// TIA Portal V16 export
// export: Created 2023-03-29T11:04:27.7848661Z, ExportSetting WithDefaults, DisplayName Totally Integrated Automation Portal, DisplayVersion V16 Update 6, DisplayName TIA Portal Version Control Interface, DisplayVersion V16 Update 2, DisplayName TIA Portal Openness, DisplayVersion V16 Update 6, DisplayName STEP 7 Professional, DisplayVersion V16 Update 6, DisplayName STEP 7 Safety, DisplayVersion V16, DisplayName WinCC Advanced, DisplayVersion V16 Update 6
ORGANIZATION_BLOCK "Startup"   // OB100, LAD, Startup
TITLE = "Complete Restart"
{ S7_Optimized_Access := 'TRUE' }
AUTHOR : RTecmer
VERSION : 0.1
// stored: AutoNumber true, IsIECCheckEnabled false, SetENOAutomatically false
   VAR_INPUT
      LostRetentive : Bool;   // True if retentive data are lost
      LostRTC : Bool;   // True if date and time are lost
   END_VAR
BEGIN

REGION Network 1: inicjacja master modbus RTU / Incjalizacja modułu Master CM1241 (RS485) Modbus RTU
   // Komunikacja z przepływomierzami MP04 i falownikiem Danfoss
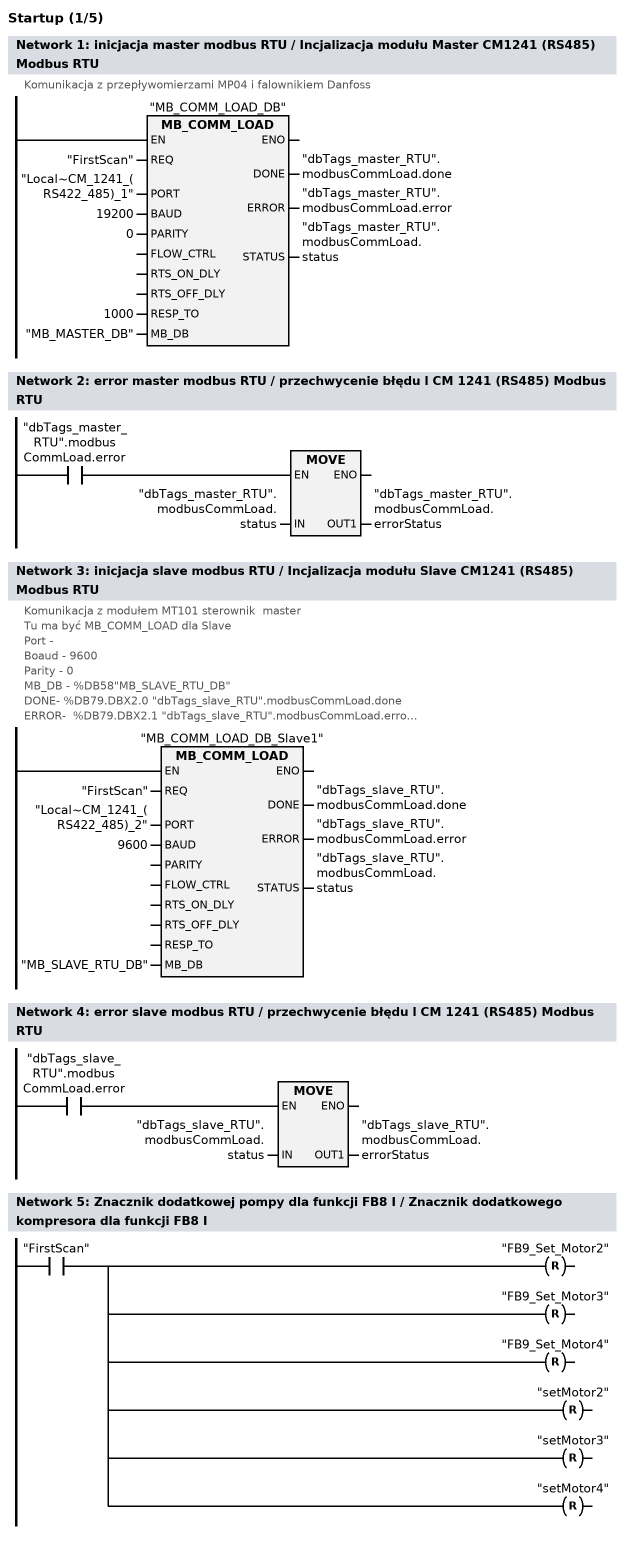
   RUNG wire#powerrail
      "MB_COMM_LOAD_DB".MB_COMM_LOAD(REQ := "FirstScan", PORT := "Local~CM_1241_(RS422_485)_1", BAUD := 19200, PARITY := 0, FLOW_CTRL :=, RTS_ON_DLY :=, RTS_OFF_DLY :=, RESP_TO := 1000, MB_DB := "MB_MASTER_DB", DONE => "dbTags_master_RTU".modbusCommLoad.done, ERROR => "dbTags_master_RTU".modbusCommLoad.error, STATUS => "dbTags_master_RTU".modbusCommLoad.status)
   END_RUNG
   // the same network as SCL:
   "MB_COMM_LOAD_DB"(REQ := "FirstScan",   // MB_COMM_LOAD
                     PORT := "Local~CM_1241_(RS422_485)_1",
                     BAUD := 19200,
                     PARITY := 0,
                     RESP_TO := 1000,
                     MB_DB := "MB_MASTER_DB",
                     DONE => "dbTags_master_RTU".modbusCommLoad.done,
                     ERROR => "dbTags_master_RTU".modbusCommLoad.error,
                     STATUS => "dbTags_master_RTU".modbusCommLoad.status);
END_REGION

REGION Network 2: error master modbus RTU / przechwycenie błędu l CM 1241 (RS485) Modbus RTU
   RUNG wire#powerrail
      Contact( "dbTags_master_RTU".modbusCommLoad.error )
      { S7_GenerateENO := "TRUE" } Move(in := "dbTags_master_RTU".modbusCommLoad.status, out1 => "dbTags_master_RTU".modbusCommLoad.errorStatus)
   END_RUNG
   // the same network as SCL:
   IF "dbTags_master_RTU".modbusCommLoad.error THEN
       "dbTags_master_RTU".modbusCommLoad.errorStatus := "dbTags_master_RTU".modbusCommLoad.status;
   END_IF;
END_REGION

REGION Network 3: inicjacja slave modbus RTU / Incjalizacja modułu Slave CM1241 (RS485) Modbus RTU
   // Komunikacja z modułem MT101 sterownik  master
   // 
   // Tu ma być MB_COMM_LOAD dla Slave
   // Port -
   // Boaud - 9600
   // Parity - 0
   // MB_DB - %DB58"MB_SLAVE_RTU_DB"
   // DONE- %DB79.DBX2.0 "dbTags_slave_RTU".modbusCommLoad.done
   // ERROR-  %DB79.DBX2.1 "dbTags_slave_RTU".modbusCommLoad.error
   // STATUS - %DB79.DBX2.2 "dbTags_slave_RTU".modbusCommLoad.status
   RUNG wire#powerrail
      "MB_COMM_LOAD_DB_Slave1".MB_COMM_LOAD(REQ := "FirstScan", PORT := "Local~CM_1241_(RS422_485)_2", BAUD := 9600, PARITY :=, FLOW_CTRL :=, RTS_ON_DLY :=, RTS_OFF_DLY :=, RESP_TO :=, MB_DB := "MB_SLAVE_RTU_DB", DONE => "dbTags_slave_RTU".modbusCommLoad.done, ERROR => "dbTags_slave_RTU".modbusCommLoad.error, STATUS => "dbTags_slave_RTU".modbusCommLoad.status)
   END_RUNG
   // the same network as SCL:
   "MB_COMM_LOAD_DB_Slave1"(REQ := "FirstScan",   // MB_COMM_LOAD
                           PORT := "Local~CM_1241_(RS422_485)_2",
                           BAUD := 9600,
                           MB_DB := "MB_SLAVE_RTU_DB",
                           DONE => "dbTags_slave_RTU".modbusCommLoad.done,
                           ERROR => "dbTags_slave_RTU".modbusCommLoad.error,
                           STATUS => "dbTags_slave_RTU".modbusCommLoad.status);
END_REGION

REGION Network 4: error slave modbus RTU / przechwycenie błędu l CM 1241 (RS485) Modbus RTU
   RUNG wire#powerrail
      Contact( "dbTags_slave_RTU".modbusCommLoad.error )
      { S7_GenerateENO := "TRUE" } Move(in := "dbTags_slave_RTU".modbusCommLoad.status, out1 => "dbTags_slave_RTU".modbusCommLoad.errorStatus)
   END_RUNG
   // the same network as SCL:
   IF "dbTags_slave_RTU".modbusCommLoad.error THEN
       "dbTags_slave_RTU".modbusCommLoad.errorStatus := "dbTags_slave_RTU".modbusCommLoad.status;
   END_IF;
END_REGION

REGION Network 5: Znacznik dodatkowej pompy dla funkcji FB8 I / Znacznik dodatkowego kompresora dla funkcji FB8 I
   RUNG wire#powerrail
      Contact( "FirstScan" )
      wire#w1
      R_Coil( "FB9_Set_Motor2" )
   END_RUNG
   RUNG wire#w1
      R_Coil( "FB9_Set_Motor3" )
   END_RUNG
   RUNG wire#w1
      R_Coil( "FB9_Set_Motor4" )
   END_RUNG
   RUNG wire#w1
      R_Coil( "setMotor2" )
   END_RUNG
   RUNG wire#w1
      R_Coil( "setMotor3" )
   END_RUNG
   RUNG wire#w1
      R_Coil( "setMotor4" )
   END_RUNG
   // the same network as SCL:
   IF "FirstScan" THEN
       "FB9_Set_Motor2" := FALSE;
       "FB9_Set_Motor3" := FALSE;
       "FB9_Set_Motor4" := FALSE;
       "setMotor2" := FALSE;
       "setMotor3" := FALSE;
       "setMotor4" := FALSE;
   END_IF;
END_REGION

REGION Network 6
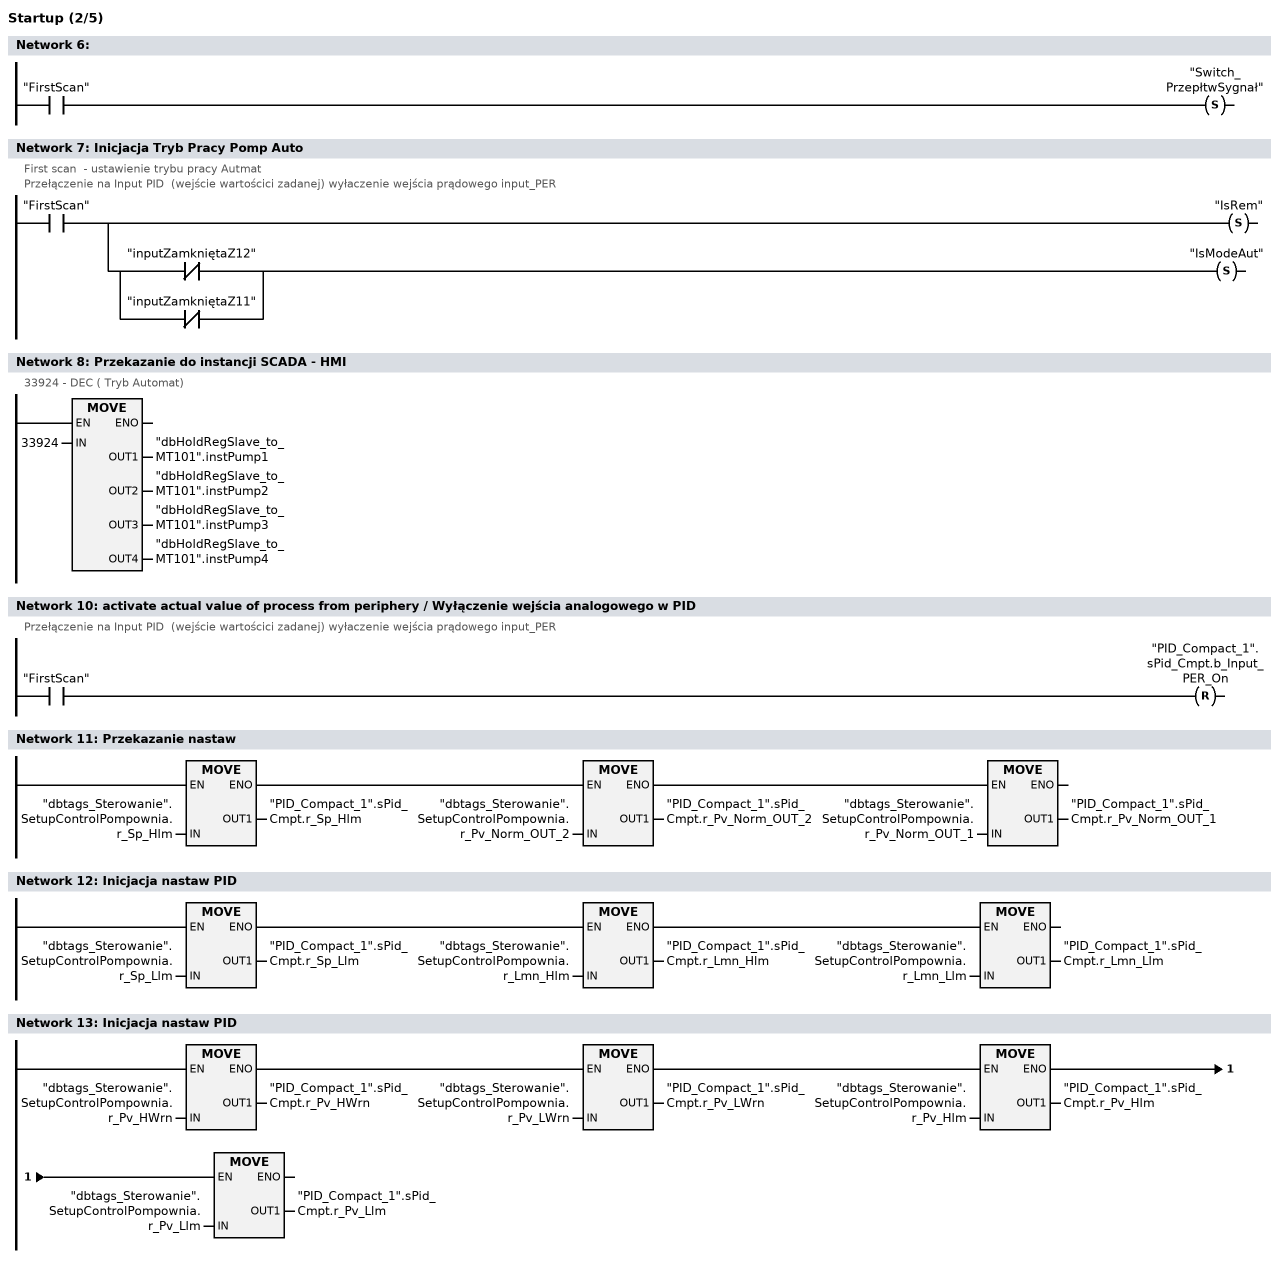
   RUNG wire#powerrail
      Contact( "FirstScan" )
      S_Coil( "Switch_PrzepłtwSygnał" )
   END_RUNG
   // the same network as SCL:
   IF "FirstScan" THEN "Switch_PrzepłtwSygnał" := TRUE; END_IF;
END_REGION

REGION Network 7: Inicjacja Tryb Pracy Pomp Auto
   // First scan  - ustawienie trybu pracy Autmat 
   // Przełączenie na Input PID  (wejście wartościci zadanej) wyłaczenie wejścia prądowego input_PER
   RUNG wire#powerrail
      Contact( "FirstScan" )
      wire#w1
      S_Coil( "IsRem" )
   END_RUNG
   RUNG wire#w1
      I_Contact( "inputZamkniętaZ12" )
      wire#w2
      S_Coil( "IsModeAut" )
   END_RUNG
   RUNG wire#w1
      I_Contact( "inputZamkniętaZ11" )
   END_RUNG wire#w2
   // the same network as SCL:
   IF "FirstScan" THEN "IsRem" := TRUE; END_IF;
   IF "FirstScan" AND (NOT "inputZamkniętaZ12" OR NOT "inputZamkniętaZ11") THEN "IsModeAut" := TRUE; END_IF;
END_REGION

REGION Network 8: Przekazanie do instancji SCADA - HMI
   // 33924 - DEC ( Tryb Automat)
   RUNG wire#powerrail
      { S7_GenerateENO := "TRUE" } Move(in := 33924, out1 => "dbHoldRegSlave_to_MT101".instPump1, out2 => "dbHoldRegSlave_to_MT101".instPump2, out3 => "dbHoldRegSlave_to_MT101".instPump3, out4 => "dbHoldRegSlave_to_MT101".instPump4)
   END_RUNG
   // the same network as SCL:
   "dbHoldRegSlave_to_MT101".instPump1 := 33924;
   "dbHoldRegSlave_to_MT101".instPump2 := 33924;
   "dbHoldRegSlave_to_MT101".instPump3 := 33924;
   "dbHoldRegSlave_to_MT101".instPump4 := 33924;
END_REGION

REGION Network 10: activate actual value of process from periphery / Wyłączenie wejścia analogowego w PID
   // Przełączenie na Input PID  (wejście wartościci zadanej) wyłaczenie wejścia prądowego input_PER
   RUNG wire#powerrail
      Contact( "FirstScan" )
      R_Coil( "PID_Compact_1".sPid_Cmpt.b_Input_PER_On )
   END_RUNG
   // the same network as SCL:
   IF "FirstScan" THEN "PID_Compact_1".sPid_Cmpt.b_Input_PER_On := FALSE; END_IF;
END_REGION

REGION Network 11: Przekazanie nastaw
   RUNG wire#powerrail
      { S7_GenerateENO := "TRUE" } Move(in := "dbtags_Sterowanie".SetupControlPompownia.r_Sp_Hlm, out1 => "PID_Compact_1".sPid_Cmpt.r_Sp_Hlm)
      { S7_GenerateENO := "TRUE" } Move(in := "dbtags_Sterowanie".SetupControlPompownia.r_Pv_Norm_OUT_2, out1 => "PID_Compact_1".sPid_Cmpt.r_Pv_Norm_OUT_2)
      { S7_GenerateENO := "TRUE" } Move(in := "dbtags_Sterowanie".SetupControlPompownia.r_Pv_Norm_OUT_1, out1 => "PID_Compact_1".sPid_Cmpt.r_Pv_Norm_OUT_1)
   END_RUNG
   // the same network as SCL:
   // ENO of a box is taken as its EN; it also drops when the box reports an error
   "PID_Compact_1".sPid_Cmpt.r_Sp_Hlm := "dbtags_Sterowanie".SetupControlPompownia.r_Sp_Hlm;
   "PID_Compact_1".sPid_Cmpt.r_Pv_Norm_OUT_2 := "dbtags_Sterowanie".SetupControlPompownia.r_Pv_Norm_OUT_2;
   "PID_Compact_1".sPid_Cmpt.r_Pv_Norm_OUT_1 := "dbtags_Sterowanie".SetupControlPompownia.r_Pv_Norm_OUT_1;
END_REGION

REGION Network 12: Inicjacja nastaw PID
   RUNG wire#powerrail
      { S7_GenerateENO := "TRUE" } Move(in := "dbtags_Sterowanie".SetupControlPompownia.r_Sp_Llm, out1 => "PID_Compact_1".sPid_Cmpt.r_Sp_Llm)
      { S7_GenerateENO := "TRUE" } Move(in := "dbtags_Sterowanie".SetupControlPompownia.r_Lmn_Hlm, out1 => "PID_Compact_1".sPid_Cmpt.r_Lmn_Hlm)
      { S7_GenerateENO := "TRUE" } Move(in := "dbtags_Sterowanie".SetupControlPompownia.r_Lmn_Llm, out1 => "PID_Compact_1".sPid_Cmpt.r_Lmn_Llm)
   END_RUNG
   // the same network as SCL:
   // ENO of a box is taken as its EN; it also drops when the box reports an error
   "PID_Compact_1".sPid_Cmpt.r_Sp_Llm := "dbtags_Sterowanie".SetupControlPompownia.r_Sp_Llm;
   "PID_Compact_1".sPid_Cmpt.r_Lmn_Hlm := "dbtags_Sterowanie".SetupControlPompownia.r_Lmn_Hlm;
   "PID_Compact_1".sPid_Cmpt.r_Lmn_Llm := "dbtags_Sterowanie".SetupControlPompownia.r_Lmn_Llm;
END_REGION

REGION Network 13: Inicjacja nastaw PID
   RUNG wire#powerrail
      { S7_GenerateENO := "TRUE" } Move(in := "dbtags_Sterowanie".SetupControlPompownia.r_Pv_HWrn, out1 => "PID_Compact_1".sPid_Cmpt.r_Pv_HWrn)
      { S7_GenerateENO := "TRUE" } Move(in := "dbtags_Sterowanie".SetupControlPompownia.r_Pv_LWrn, out1 => "PID_Compact_1".sPid_Cmpt.r_Pv_LWrn)
      { S7_GenerateENO := "TRUE" } Move(in := "dbtags_Sterowanie".SetupControlPompownia.r_Pv_Hlm, out1 => "PID_Compact_1".sPid_Cmpt.r_Pv_Hlm)
      { S7_GenerateENO := "TRUE" } Move(in := "dbtags_Sterowanie".SetupControlPompownia.r_Pv_Llm, out1 => "PID_Compact_1".sPid_Cmpt.r_Pv_Llm)
   END_RUNG
   // the same network as SCL:
   // ENO of a box is taken as its EN; it also drops when the box reports an error
   "PID_Compact_1".sPid_Cmpt.r_Pv_HWrn := "dbtags_Sterowanie".SetupControlPompownia.r_Pv_HWrn;
   "PID_Compact_1".sPid_Cmpt.r_Pv_LWrn := "dbtags_Sterowanie".SetupControlPompownia.r_Pv_LWrn;
   "PID_Compact_1".sPid_Cmpt.r_Pv_Hlm := "dbtags_Sterowanie".SetupControlPompownia.r_Pv_Hlm;
   "PID_Compact_1".sPid_Cmpt.r_Pv_Llm := "dbtags_Sterowanie".SetupControlPompownia.r_Pv_Llm;
END_REGION

REGION Network 14: Zasuwa Z11 Tryb Automat
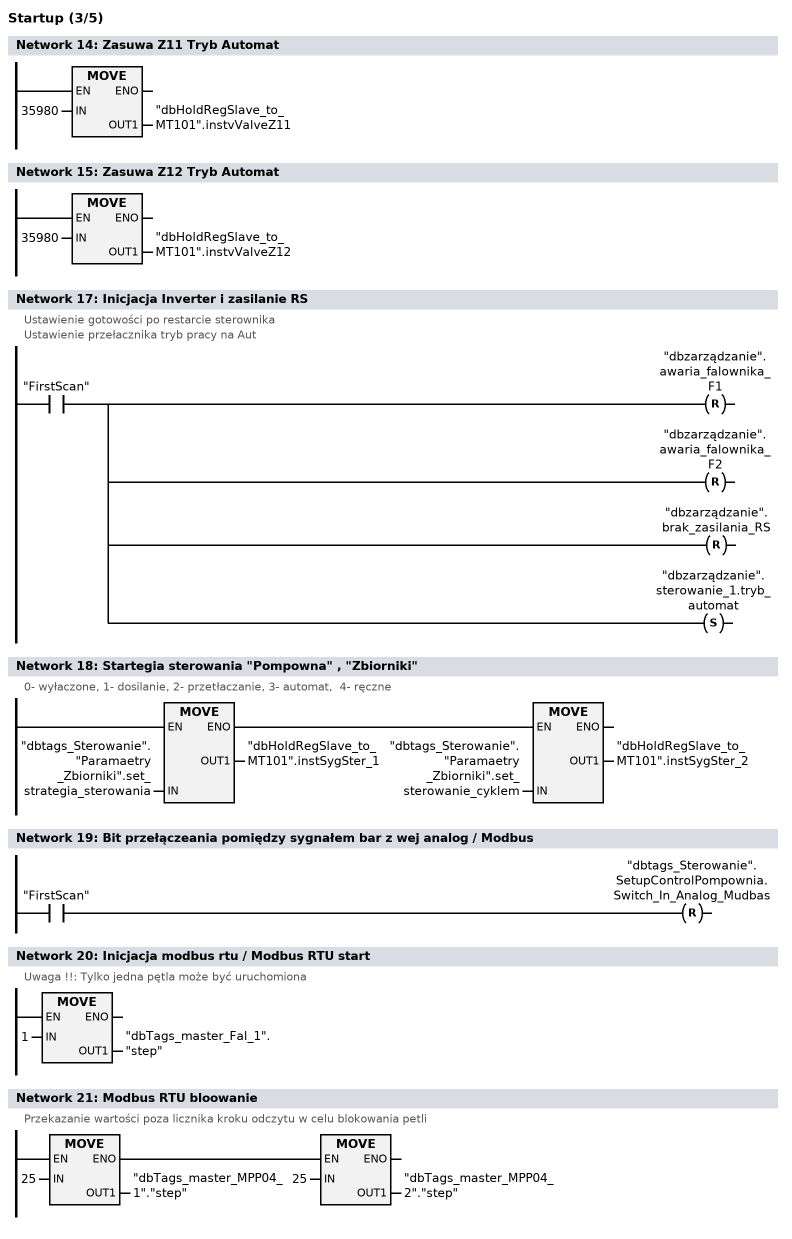
   RUNG wire#powerrail
      Move(in := 35980, out1 => "dbHoldRegSlave_to_MT101".instvValveZ11)
   END_RUNG
   // the same network as SCL:
   "dbHoldRegSlave_to_MT101".instvValveZ11 := 35980;
END_REGION

REGION Network 15: Zasuwa Z12 Tryb Automat
   RUNG wire#powerrail
      Move(in := 35980, out1 => "dbHoldRegSlave_to_MT101".instvValveZ12)
   END_RUNG
   // the same network as SCL:
   "dbHoldRegSlave_to_MT101".instvValveZ12 := 35980;
END_REGION

REGION Network 17: Inicjacja Inverter i zasilanie RS
   // Ustawienie gotowości po restarcie sterownika
   // Ustawienie przełacznika tryb pracy na Aut
   RUNG wire#powerrail
      Contact( "FirstScan" )
      wire#w1
      R_Coil( "dbzarządzanie".awaria_falownika_F1 )
   END_RUNG
   RUNG wire#w1
      R_Coil( "dbzarządzanie".awaria_falownika_F2 )
   END_RUNG
   RUNG wire#w1
      R_Coil( "dbzarządzanie".brak_zasilania_RS )
   END_RUNG
   RUNG wire#w1
      S_Coil( "dbzarządzanie".sterowanie_1.tryb_automat )
   END_RUNG
   // the same network as SCL:
   IF "FirstScan" THEN
       "dbzarządzanie".awaria_falownika_F1 := FALSE;
       "dbzarządzanie".awaria_falownika_F2 := FALSE;
       "dbzarządzanie".brak_zasilania_RS := FALSE;
       "dbzarządzanie".sterowanie_1.tryb_automat := TRUE;
   END_IF;
END_REGION

REGION Network 18: Startegia sterowania "Pompowna" , "Zbiorniki"
   // 0- wyłaczone, 1- dosilanie, 2- przetłaczanie, 3- automat,  4- ręczne
   RUNG wire#powerrail
      Move(in := "dbtags_Sterowanie"."Paramaetry _Zbiorniki".set_strategia_sterowania, out1 => "dbHoldRegSlave_to_MT101".instSygSter_1)
      Move(in := "dbtags_Sterowanie"."Paramaetry _Zbiorniki".set_sterowanie_cyklem, out1 => "dbHoldRegSlave_to_MT101".instSygSter_2)
   END_RUNG
   // the same network as SCL:
   "dbHoldRegSlave_to_MT101".instSygSter_1 := "dbtags_Sterowanie"."Paramaetry _Zbiorniki".set_strategia_sterowania;
   "dbHoldRegSlave_to_MT101".instSygSter_2 := "dbtags_Sterowanie"."Paramaetry _Zbiorniki".set_sterowanie_cyklem;
END_REGION

REGION Network 19: Bit przełączeania pomiędzy sygnałem bar z wej analog / Modbus
   RUNG wire#powerrail
      Contact( "FirstScan" )
      R_Coil( "dbtags_Sterowanie".SetupControlPompownia.Switch_In_Analog_Mudbas )
   END_RUNG
   // the same network as SCL:
   IF "FirstScan" THEN "dbtags_Sterowanie".SetupControlPompownia.Switch_In_Analog_Mudbas := FALSE; END_IF;
END_REGION

REGION Network 20: Inicjacja modbus rtu / Modbus RTU start
   // Uwaga !!: Tylko jedna pętla może być uruchomiona
   RUNG wire#powerrail
      { S7_GenerateENO := "TRUE" } Move(in := 1, out1 => "dbTags_master_Fal_1"."step")
   END_RUNG
   // the same network as SCL:
   "dbTags_master_Fal_1"."step" := 1;
END_REGION

REGION Network 21: Modbus RTU bloowanie
   // Przekazanie wartości poza licznika kroku odczytu w celu blokowania petli
   RUNG wire#powerrail
      { S7_GenerateENO := "TRUE" } Move(in := 25, out1 => "dbTags_master_MPP04_1"."step")
      { S7_GenerateENO := "TRUE" } Move(in := 25, out1 => "dbTags_master_MPP04_2"."step")
   END_RUNG
   // the same network as SCL:
   // ENO of a box is taken as its EN; it also drops when the box reports an error
   "dbTags_master_MPP04_1"."step" := 25;
   "dbTags_master_MPP04_2"."step" := 25;
END_REGION

REGION Network 22: Przełącznik wyboru źródła zadawania wartości granicznej dopuszczalnego prądy falownika
   // 1 - zadawany w konfiguracju z HMI
   // 0 - odczytany z falownika
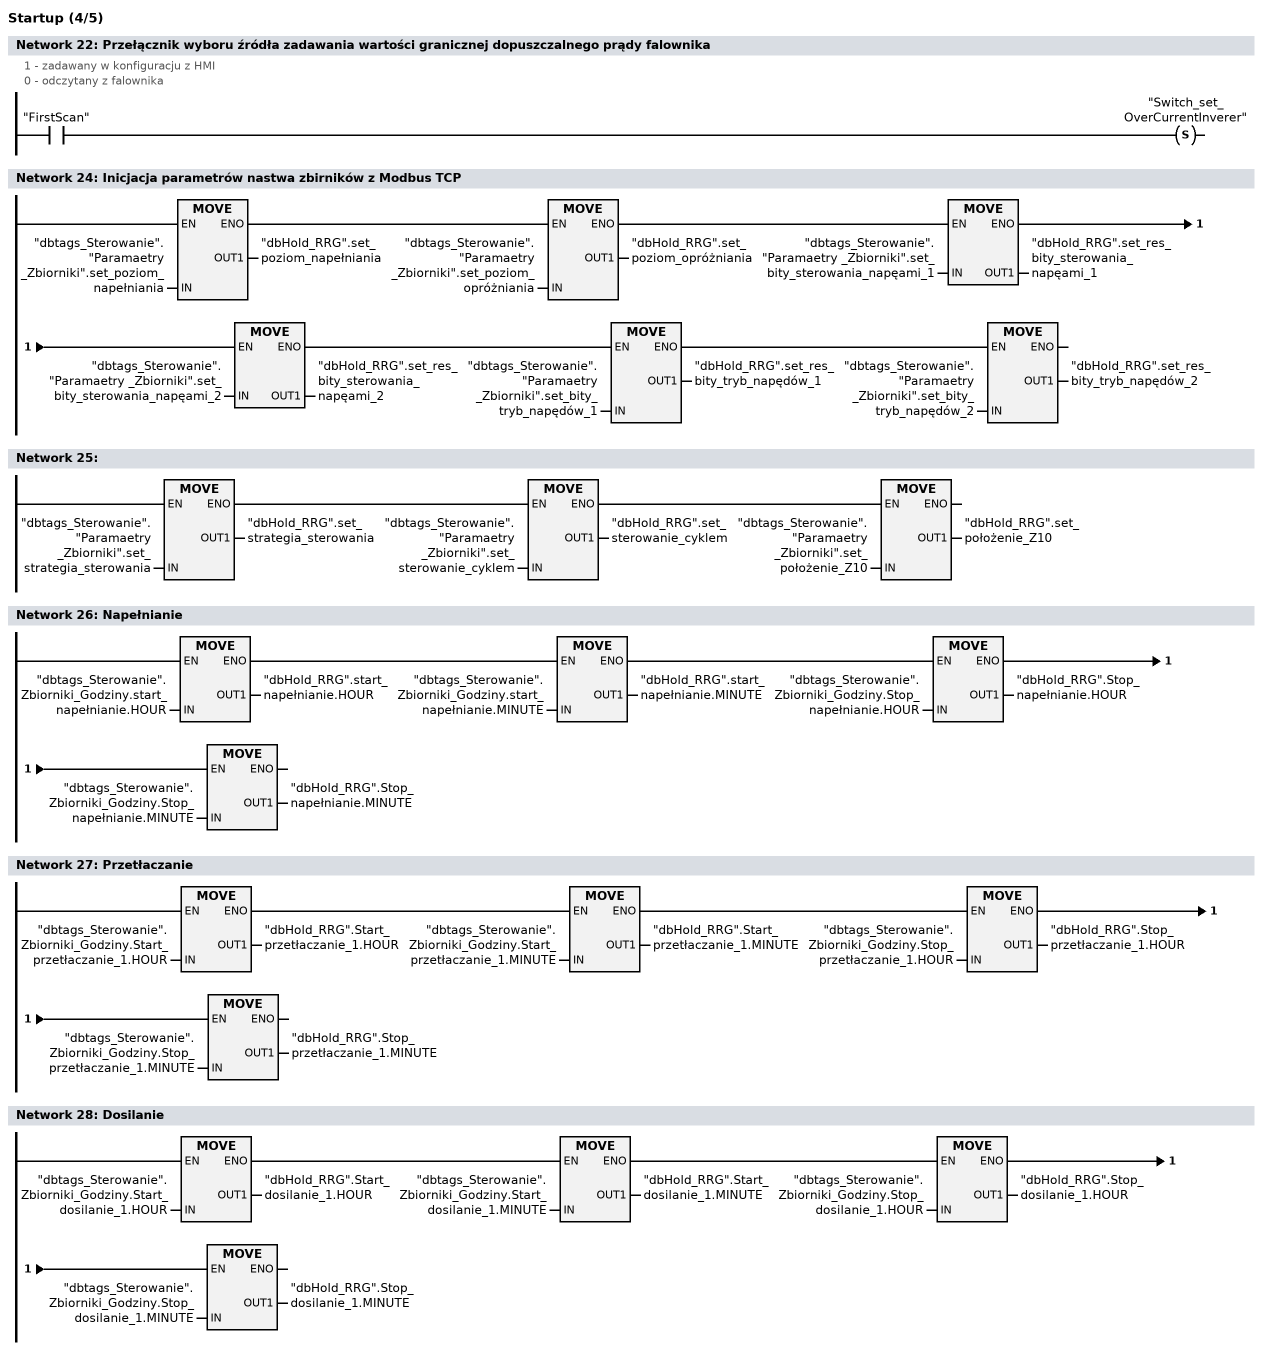
   RUNG wire#powerrail
      Contact( "FirstScan" )
      S_Coil( "Switch_set_OverCurrentInverer" )
   END_RUNG
   // the same network as SCL:
   IF "FirstScan" THEN "Switch_set_OverCurrentInverer" := TRUE; END_IF;
END_REGION

REGION Network 23 (SCL): Ustawienie Setpoint SV do regulatora
   // Wartość ciśnienia zadanego zależna od wybranej strategii
   CASE "dbHoldRegSlave_to_MT101".instSygSter_1 OF
     1:
       "dbdane".Setpoint_SV := "dbtags_Sterowanie".SetupControlPompownia.set_barDN500_B5 ;
     2:
       "dbdane".Setpoint_SV := "dbtags_Sterowanie".SetupControlPompownia.set_barDN225_B6;
     3:
       "dbdane".Setpoint_SV := "dbdane".Setpoint_bar_automat ;

     ELSE
       "dbdane".Setpoint_SV := 0.0;
       ;
   END_CASE;
END_REGION

REGION Network 24: Inicjacja parametrów nastwa zbirników z Modbus TCP
   RUNG wire#powerrail
      Move(in := "dbtags_Sterowanie"."Paramaetry _Zbiorniki".set_poziom_napełniania, out1 => "dbHold_RRG".set_poziom_napełniania)
      Move(in := "dbtags_Sterowanie"."Paramaetry _Zbiorniki".set_poziom_opróżniania, out1 => "dbHold_RRG".set_poziom_opróżniania)
      Move(in := "dbtags_Sterowanie"."Paramaetry _Zbiorniki".set_bity_sterowania_napęami_1, out1 => "dbHold_RRG".set_res_bity_sterowania_napęami_1)
      Move(in := "dbtags_Sterowanie"."Paramaetry _Zbiorniki".set_bity_sterowania_napęami_2, out1 => "dbHold_RRG".set_res_bity_sterowania_napęami_2)
      Move(in := "dbtags_Sterowanie"."Paramaetry _Zbiorniki".set_bity_tryb_napędów_1, out1 => "dbHold_RRG".set_res_bity_tryb_napędów_1)
      Move(in := "dbtags_Sterowanie"."Paramaetry _Zbiorniki".set_bity_tryb_napędów_2, out1 => "dbHold_RRG".set_res_bity_tryb_napędów_2)
   END_RUNG
   // the same network as SCL:
   "dbHold_RRG".set_poziom_napełniania := "dbtags_Sterowanie"."Paramaetry _Zbiorniki".set_poziom_napełniania;
   "dbHold_RRG".set_poziom_opróżniania := "dbtags_Sterowanie"."Paramaetry _Zbiorniki".set_poziom_opróżniania;
   "dbHold_RRG".set_res_bity_sterowania_napęami_1 := "dbtags_Sterowanie"."Paramaetry _Zbiorniki".set_bity_sterowania_napęami_1;
   "dbHold_RRG".set_res_bity_sterowania_napęami_2 := "dbtags_Sterowanie"."Paramaetry _Zbiorniki".set_bity_sterowania_napęami_2;
   "dbHold_RRG".set_res_bity_tryb_napędów_1 := "dbtags_Sterowanie"."Paramaetry _Zbiorniki".set_bity_tryb_napędów_1;
   "dbHold_RRG".set_res_bity_tryb_napędów_2 := "dbtags_Sterowanie"."Paramaetry _Zbiorniki".set_bity_tryb_napędów_2;
END_REGION

REGION Network 25
   RUNG wire#powerrail
      Move(in := "dbtags_Sterowanie"."Paramaetry _Zbiorniki".set_strategia_sterowania, out1 => "dbHold_RRG".set_strategia_sterowania)
      Move(in := "dbtags_Sterowanie"."Paramaetry _Zbiorniki".set_sterowanie_cyklem, out1 => "dbHold_RRG".set_sterowanie_cyklem)
      Move(in := "dbtags_Sterowanie"."Paramaetry _Zbiorniki".set_położenie_Z10, out1 => "dbHold_RRG".set_położenie_Z10)
   END_RUNG
   // the same network as SCL:
   "dbHold_RRG".set_strategia_sterowania := "dbtags_Sterowanie"."Paramaetry _Zbiorniki".set_strategia_sterowania;
   "dbHold_RRG".set_sterowanie_cyklem := "dbtags_Sterowanie"."Paramaetry _Zbiorniki".set_sterowanie_cyklem;
   "dbHold_RRG".set_położenie_Z10 := "dbtags_Sterowanie"."Paramaetry _Zbiorniki".set_położenie_Z10;
END_REGION

REGION Network 26: Napełnianie
   RUNG wire#powerrail
      Move(in := "dbtags_Sterowanie".Zbiorniki_Godziny.start_napełnianie.HOUR, out1 => "dbHold_RRG".start_napełnianie.HOUR)
      Move(in := "dbtags_Sterowanie".Zbiorniki_Godziny.start_napełnianie.MINUTE, out1 => "dbHold_RRG".start_napełnianie.MINUTE)
      Move(in := "dbtags_Sterowanie".Zbiorniki_Godziny.Stop_napełnianie.HOUR, out1 => "dbHold_RRG".Stop_napełnianie.HOUR)
      Move(in := "dbtags_Sterowanie".Zbiorniki_Godziny.Stop_napełnianie.MINUTE, out1 => "dbHold_RRG".Stop_napełnianie.MINUTE)
   END_RUNG
   // the same network as SCL:
   "dbHold_RRG".start_napełnianie.HOUR := "dbtags_Sterowanie".Zbiorniki_Godziny.start_napełnianie.HOUR;
   "dbHold_RRG".start_napełnianie.MINUTE := "dbtags_Sterowanie".Zbiorniki_Godziny.start_napełnianie.MINUTE;
   "dbHold_RRG".Stop_napełnianie.HOUR := "dbtags_Sterowanie".Zbiorniki_Godziny.Stop_napełnianie.HOUR;
   "dbHold_RRG".Stop_napełnianie.MINUTE := "dbtags_Sterowanie".Zbiorniki_Godziny.Stop_napełnianie.MINUTE;
END_REGION

REGION Network 27: Przetłaczanie
   RUNG wire#powerrail
      Move(in := "dbtags_Sterowanie".Zbiorniki_Godziny.Start_przetłaczanie_1.HOUR, out1 => "dbHold_RRG".Start_przetłaczanie_1.HOUR)
      Move(in := "dbtags_Sterowanie".Zbiorniki_Godziny.Start_przetłaczanie_1.MINUTE, out1 => "dbHold_RRG".Start_przetłaczanie_1.MINUTE)
      Move(in := "dbtags_Sterowanie".Zbiorniki_Godziny.Stop_przetłaczanie_1.HOUR, out1 => "dbHold_RRG".Stop_przetłaczanie_1.HOUR)
      Move(in := "dbtags_Sterowanie".Zbiorniki_Godziny.Stop_przetłaczanie_1.MINUTE, out1 => "dbHold_RRG".Stop_przetłaczanie_1.MINUTE)
   END_RUNG
   // the same network as SCL:
   "dbHold_RRG".Start_przetłaczanie_1.HOUR := "dbtags_Sterowanie".Zbiorniki_Godziny.Start_przetłaczanie_1.HOUR;
   "dbHold_RRG".Start_przetłaczanie_1.MINUTE := "dbtags_Sterowanie".Zbiorniki_Godziny.Start_przetłaczanie_1.MINUTE;
   "dbHold_RRG".Stop_przetłaczanie_1.HOUR := "dbtags_Sterowanie".Zbiorniki_Godziny.Stop_przetłaczanie_1.HOUR;
   "dbHold_RRG".Stop_przetłaczanie_1.MINUTE := "dbtags_Sterowanie".Zbiorniki_Godziny.Stop_przetłaczanie_1.MINUTE;
END_REGION

REGION Network 28: Dosilanie
   RUNG wire#powerrail
      Move(in := "dbtags_Sterowanie".Zbiorniki_Godziny.Start_dosilanie_1.HOUR, out1 => "dbHold_RRG".Start_dosilanie_1.HOUR)
      Move(in := "dbtags_Sterowanie".Zbiorniki_Godziny.Start_dosilanie_1.MINUTE, out1 => "dbHold_RRG".Start_dosilanie_1.MINUTE)
      Move(in := "dbtags_Sterowanie".Zbiorniki_Godziny.Stop_dosilanie_1.HOUR, out1 => "dbHold_RRG".Stop_dosilanie_1.HOUR)
      Move(in := "dbtags_Sterowanie".Zbiorniki_Godziny.Stop_dosilanie_1.MINUTE, out1 => "dbHold_RRG".Stop_dosilanie_1.MINUTE)
   END_RUNG
   // the same network as SCL:
   "dbHold_RRG".Start_dosilanie_1.HOUR := "dbtags_Sterowanie".Zbiorniki_Godziny.Start_dosilanie_1.HOUR;
   "dbHold_RRG".Start_dosilanie_1.MINUTE := "dbtags_Sterowanie".Zbiorniki_Godziny.Start_dosilanie_1.MINUTE;
   "dbHold_RRG".Stop_dosilanie_1.HOUR := "dbtags_Sterowanie".Zbiorniki_Godziny.Stop_dosilanie_1.HOUR;
   "dbHold_RRG".Stop_dosilanie_1.MINUTE := "dbtags_Sterowanie".Zbiorniki_Godziny.Stop_dosilanie_1.MINUTE;
END_REGION

REGION Network 29: załącz/ wyłą filtrowanie przez kolmana analogów
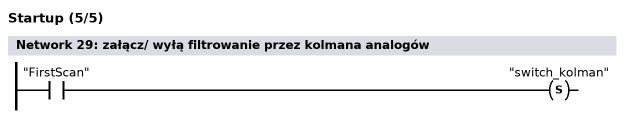
   RUNG wire#powerrail
      Contact( "FirstScan" )
      S_Coil( "switch_kolman" )
   END_RUNG
   // the same network as SCL:
   IF "FirstScan" THEN "switch_kolman" := TRUE; END_IF;
END_REGION
END_ORGANIZATION_BLOCK
